{attribute 'qualified_only'}
VAR_GLOBAL CONSTANT
(* Super Mario Brothers Overworld *)
	NOTES_MAX : UINT := 3324;
	notes : ARRAY[0..NOTES_MAX] OF REAL := [146, 20, 0, 369, 20, 0, 659, 20, 47, 146, 20, 0, 369, 20, 0, 659, 20, 189, 146, 20, 0, 369, 20, 0, 659, 20, 190, 146, 20, 0, 369, 20, 0, 523, 20, 47, 146, 20, 0, 369, 20, 0, 659, 20, 190, 391, 20, 0, 493, 20, 0, 783, 20, 475, 195, 20, 0, 391, 20, 0, 195, 20, 0, 391, 20, 473, 195, 20, 0, 329, 20, 0, 523, 20, 332, 164, 20, 0, 261, 20, 0, 391, 20, 332, 130, 20, 0, 195, 20, 0, 329, 20, 332, 174, 20, 0, 261, 20, 0, 440, 20, 189, 195, 20, 0, 293, 20, 0, 493, 20, 189, 184, 20, 0, 277, 20, 0, 466, 20, 47, 174, 20, 0, 261, 20, 0, 440, 20, 190, 164, 20, 0, 261, 20, 0, 391, 20, 95, 261, 20, 0, 391, 20, 0, 659, 20, 95, 329, 20, 0, 493, 20, 0, 783, 20, 95, 349, 20, 0, 523, 20, 0, 880, 20, 190, 293, 20, 0, 440, 20, 0, 698, 20, 47, 329, 20, 0, 493, 20, 0, 783, 20, 189, 261, 20, 0, 440, 20, 0, 659, 20, 189, 220, 20, 0, 329, 20, 0, 523, 20, 47, 246, 20, 0, 349, 20, 0, 587, 20, 47, 195, 20, 0, 293, 20, 0, 493, 20, 332, 195, 20, 0, 329, 20, 0, 523, 20, 332, 164, 20, 0, 261, 20, 0, 391, 20, 332, 130, 20, 0, 195, 20, 0, 329, 20, 332, 174, 20, 0, 261, 20, 0, 440, 20, 189, 195, 20, 0, 293, 20, 0, 493, 20, 189, 184, 20, 0, 277, 20, 0, 466, 20, 47, 174, 20, 0, 261, 20, 0, 440, 20, 190, 164, 20, 0, 261, 20, 0, 391, 20, 95, 261, 20, 0, 391, 20, 0, 659, 20, 95, 329, 20, 0, 493, 20, 0, 783, 20, 95, 349, 20, 0, 523, 20, 0, 880, 20, 190, 293, 20, 0, 440, 20, 0, 698, 20, 47, 329, 20, 0, 493, 20, 0, 783, 20, 189, 261, 20, 0, 440, 20, 0, 659, 20, 189, 220, 20, 0, 329, 20, 0, 523, 20, 47, 246, 20, 0, 349, 20, 0, 587, 20, 47, 195, 20, 0, 293, 20, 0, 493, 20, 332, 130, 95, 190, 659, 20, 0, 783, 20, 0, 659, 20, 0, 783, 20, 47, 195, 20, 0, 622, 20, 0, 739, 20, 47, 587, 20, 0, 698, 20, 0, 587, 20, 0, 698, 20, 47, 493, 20, 0, 622, 20, 0, 493, 20, 0, 622, 20, 47, 261, 95, 47, 523, 20, 0, 659, 20, 0, 523, 20, 0, 659, 20, 47, 174, 95, 47, 329, 20, 0, 415, 20, 0, 329, 20, 0, 415, 20, 47, 349, 20, 0, 440, 20, 0, 349, 20, 0, 440, 20, 47, 261, 20, 0, 391, 20, 0, 523, 20, 47, 261, 95, 47, 261, 20, 0, 440, 20, 0, 261, 20, 0, 440, 20, 47, 174, 20, 0, 329, 20, 0, 523, 20, 47, 349, 20, 0, 587, 20, 0, 349, 20, 0, 587, 20, 47, 130, 95, 190, 659, 20, 0, 783, 20, 0, 659, 20, 0, 783, 20, 47, 164, 20, 0, 622, 20, 0, 739, 20, 47, 587, 20, 0, 698, 20, 0, 587, 20, 0, 698, 20, 47, 493, 20, 0, 622, 20, 0, 493, 20, 0, 622, 20, 47, 195, 95, 47, 261, 20, 0, 523, 20, 0, 659, 20, 189, 698, 20, 0, 783, 20, 0, 1046, 20, 189, 698, 20, 0, 783, 20, 0, 1046, 20, 47, 698, 20, 0, 783, 20, 0, 1046, 20, 190, 195, 95, 190, 130, 95, 190, 659, 20, 0, 783, 20, 0, 659, 20, 0, 783, 20, 47, 195, 20, 0, 622, 20, 0, 739, 20, 47, 587, 20, 0, 698, 20, 0, 587, 20, 0, 698, 20, 47, 493, 20, 0, 622, 20, 0, 493, 20, 0, 622, 20, 47, 261, 95, 47, 523, 20, 0, 659, 20, 0, 523, 20, 0, 659, 20, 47, 174, 95, 47, 329, 20, 0, 415, 20, 0, 329, 20, 0, 415, 20, 47, 349, 20, 0, 440, 20, 0, 349, 20, 0, 440, 20, 47, 261, 20, 0, 391, 20, 0, 523, 20, 47, 261, 95, 47, 261, 20, 0, 440, 20, 0, 261, 20, 0, 440, 20, 47, 174, 20, 0, 329, 20, 0, 523, 20, 47, 349, 20, 0, 587, 20, 0, 349, 20, 0, 587, 20, 47, 130, 95, 190, 207, 20, 0, 415, 20, 0, 622, 20, 332, 233, 20, 0, 349, 20, 0, 587, 20, 332, 261, 20, 0, 329, 20, 0, 523, 20, 332, 195, 94, 47, 195, 95, 190, 130, 95, 190, 130, 95, 190, 659, 20, 0, 783, 20, 0, 659, 20, 0, 783, 20, 47, 195, 20, 0, 622, 20, 0, 739, 20, 47, 587, 20, 0, 698, 20, 0, 587, 20, 0, 698, 20, 47, 493, 20, 0, 622, 20, 0, 493, 20, 0, 622, 20, 47, 261, 95, 47, 523, 20, 0, 659, 20, 0, 523, 20, 0, 659, 20, 47, 174, 95, 47, 329, 20, 0, 415, 20, 0, 329, 20, 0, 415, 20, 47, 349, 20, 0, 440, 20, 0, 349, 20, 0, 440, 20, 47, 261, 20, 0, 391, 20, 0, 523, 20, 47, 261, 95, 47, 261, 20, 0, 440, 20, 0, 261, 20, 0, 440, 20, 47, 174, 20, 0, 329, 20, 0, 523, 20, 47, 349, 20, 0, 587, 20, 0, 349, 20, 0, 587, 20, 47, 130, 95, 190, 659, 20, 0, 783, 20, 0, 659, 20, 0, 783, 20, 47, 164, 20, 0, 622, 20, 0, 739, 20, 47, 587, 20, 0, 698, 20, 0, 587, 20, 0, 698, 20, 47, 493, 20, 0, 622, 20, 0, 493, 20, 0, 622, 20, 47, 195, 95, 47, 261, 20, 0, 523, 20, 0, 659, 20, 189, 698, 20, 0, 783, 20, 0, 1046, 20, 189, 698, 20, 0, 783, 20, 0, 1046, 20, 47, 698, 20, 0, 783, 20, 0, 1046, 20, 190, 195, 95, 190, 130, 95, 190, 659, 20, 0, 783, 20, 0, 659, 20, 0, 783, 20, 47, 195, 20, 0, 622, 20, 0, 739, 20, 47, 587, 20, 0, 698, 20, 0, 587, 20, 0, 698, 20, 47, 493, 20, 0, 622, 20, 0, 493, 20, 0, 622, 20, 47, 261, 95, 47, 523, 20, 0, 659, 20, 0, 523, 20, 0, 659, 20, 47, 174, 95, 47, 329, 20, 0, 415, 20, 0, 329, 20, 0, 415, 20, 47, 349, 20, 0, 440, 20, 0, 349, 20, 0, 440, 20, 47, 261, 20, 0, 391, 20, 0, 523, 20, 47, 261, 95, 47, 261, 20, 0, 440, 20, 0, 261, 20, 0, 440, 20, 47, 174, 20, 0, 329, 20, 0, 523, 20, 47, 349, 20, 0, 587, 20, 0, 349, 20, 0, 587, 20, 47, 130, 95, 190, 207, 20, 0, 415, 20, 0, 622, 20, 332, 233, 20, 0, 349, 20, 0, 587, 20, 332, 261, 20, 0, 329, 20, 0, 523, 20, 332, 195, 94, 47, 195, 95, 190, 130, 95, 190, 103, 20, 0, 415, 20, 0, 523, 20, 47, 415, 20, 0, 523, 20, 0, 415, 20, 0, 523, 20, 189, 155, 20, 0, 415, 20, 0, 523, 20, 190, 415, 20, 0, 523, 20, 0, 415, 20, 0, 523, 20, 47, 207, 20, 0, 466, 20, 0, 587, 20, 190, 195, 20, 0, 391, 20, 0, 659, 20, 47, 329, 20, 0, 523, 20, 0, 329, 20, 0, 523, 20, 190, 130, 20, 0, 329, 20, 0, 440, 20, 47, 261, 20, 0, 391, 20, 0, 261, 20, 0, 391, 20, 189, 97, 95, 189, 103, 20, 0, 415, 20, 0, 523, 20, 47, 415, 20, 0, 523, 20, 0, 415, 20, 0, 523, 20, 189, 155, 20, 0, 415, 20, 0, 523, 20, 190, 415, 20, 0, 523, 20, 0, 415, 20, 0, 523, 20, 47, 207, 20, 0, 466, 20, 0, 587, 20, 47, 391, 20, 0, 659, 20, 0, 391, 20, 0, 659, 20, 47, 195, 95, 333, 130, 95, 332, 97, 95, 189, 103, 20, 0, 415, 20, 0, 523, 20, 47, 415, 20, 0, 523, 20, 0, 415, 20, 0, 523, 20, 189, 155, 20, 0, 415, 20, 0, 523, 20, 190, 415, 20, 0, 523, 20, 0, 415, 20, 0, 523, 20, 47, 207, 20, 0, 466, 20, 0, 587, 20, 190, 195, 20, 0, 391, 20, 0, 659, 20, 47, 329, 20, 0, 523, 20, 0, 329, 20, 0, 523, 20, 190, 130, 20, 0, 329, 20, 0, 440, 20, 47, 261, 20, 0, 391, 20, 0, 261, 20, 0, 391, 20, 189, 97, 95, 189, 146, 20, 0, 369, 20, 0, 659, 20, 47, 146, 20, 0, 369, 20, 0, 659, 20, 189, 146, 20, 0, 369, 20, 0, 659, 20, 190, 146, 20, 0, 369, 20, 0, 523, 20, 47, 146, 20, 0, 369, 20, 0, 659, 20, 190, 391, 20, 0, 493, 20, 0, 783, 20, 475, 195, 20, 0, 391, 20, 0, 195, 20, 0, 391, 20, 473, 195, 20, 0, 329, 20, 0, 523, 20, 332, 164, 20, 0, 261, 20, 0, 391, 20, 332, 130, 20, 0, 195, 20, 0, 329, 20, 332, 174, 20, 0, 261, 20, 0, 440, 20, 189, 195, 20, 0, 293, 20, 0, 493, 20, 189, 184, 20, 0, 277, 20, 0, 466, 20, 47, 174, 20, 0, 261, 20, 0, 440, 20, 190, 164, 20, 0, 261, 20, 0, 391, 20, 95, 261, 20, 0, 391, 20, 0, 659, 20, 95, 329, 20, 0, 493, 20, 0, 783, 20, 95, 349, 20, 0, 523, 20, 0, 880, 20, 190, 293, 20, 0, 440, 20, 0, 698, 20, 47, 329, 20, 0, 493, 20, 0, 783, 20, 189, 261, 20, 0, 440, 20, 0, 659, 20, 189, 220, 20, 0, 329, 20, 0, 523, 20, 47, 246, 20, 0, 349, 20, 0, 587, 20, 47, 195, 20, 0, 293, 20, 0, 493, 20, 332, 195, 20, 0, 329, 20, 0, 523, 20, 332, 164, 20, 0, 261, 20, 0, 391, 20, 332, 130, 20, 0, 195, 20, 0, 329, 20, 332, 174, 20, 0, 261, 20, 0, 440, 20, 189, 195, 20, 0, 293, 20, 0, 493, 20, 189, 184, 20, 0, 277, 20, 0, 466, 20, 47, 174, 20, 0, 261, 20, 0, 440, 20, 190, 164, 20, 0, 261, 20, 0, 391, 20, 95, 261, 20, 0, 391, 20, 0, 659, 20, 95, 329, 20, 0, 493, 20, 0, 783, 20, 95, 349, 20, 0, 523, 20, 0, 880, 20, 190, 293, 20, 0, 440, 20, 0, 698, 20, 47, 329, 20, 0, 493, 20, 0, 783, 20, 189, 261, 20, 0, 440, 20, 0, 659, 20, 189, 220, 20, 0, 329, 20, 0, 523, 20, 47, 246, 20, 0, 349, 20, 0, 587, 20, 47, 195, 20, 0, 293, 20, 0, 493, 20, 332, 130, 20, 0, 523, 20, 0, 659, 20, 47, 440, 20, 0, 523, 20, 0, 440, 20, 0, 523, 20, 190, 184, 20, 0, 329, 20, 0, 391, 20, 47, 195, 95, 190, 261, 20, 0, 329, 20, 0, 415, 20, 190, 174, 20, 0, 349, 20, 0, 440, 20, 47, 523, 20, 0, 698, 20, 0, 523, 20, 0, 698, 20, 47, 174, 95, 47, 523, 20, 0, 698, 20, 0, 523, 20, 0, 698, 20, 47, 261, 20, 0, 349, 20, 0, 440, 20, 47, 261, 94, 47, 174, 95, 190, 146, 20, 0, 391, 20, 0, 493, 20, 95, 698, 20, 0, 880, 20, 0, 698, 20, 0, 880, 20, 95, 698, 20, 0, 880, 20, 0, 174, 15, 0, 698, 15, 0, 880, 15, 0, 174, 47, 47, 195, 20, 0, 698, 20, 0, 880, 20, 95, 659, 20, 0, 783, 20, 0, 659, 20, 0, 783, 20, 0, 246, 95, 0, 587, 20, 0, 698, 20, 0, 587, 20, 0, 698, 20, 95, 195, 20, 0, 523, 20, 0, 659, 20, 47, 440, 20, 0, 523, 20, 0, 440, 20, 0, 523, 20, 47, 195, 95, 47, 349, 20, 0, 440, 20, 0, 349, 20, 0, 440, 20, 47, 261, 20, 0, 329, 20, 0, 391, 20, 47, 261, 94, 47, 195, 95, 190, 130, 20, 0, 523, 20, 0, 659, 20, 47, 440, 20, 0, 523, 20, 0, 440, 20, 0, 523, 20, 190, 184, 20, 0, 329, 20, 0, 391, 20, 47, 195, 95, 190, 261, 20, 0, 329, 20, 0, 415, 20, 190, 174, 20, 0, 349, 20, 0, 440, 20, 47, 523, 20, 0, 698, 20, 0, 523, 20, 0, 698, 20, 47, 174, 95, 47, 523, 20, 0, 698, 20, 0, 523, 20, 0, 698, 20, 47, 261, 20, 0, 349, 20, 0, 440, 20, 47, 261, 94, 47, 174, 95, 190, 195, 20, 0, 391, 20, 0, 493, 20, 47, 195, 20, 0, 587, 20, 0, 698, 20, 190, 195, 20, 0, 587, 20, 0, 698, 20, 47, 195, 20, 0, 587, 20, 0, 698, 20, 95, 220, 20, 0, 523, 20, 0, 659, 20, 95, 246, 20, 0, 493, 20, 0, 587, 20, 95, 261, 20, 0, 391, 20, 0, 523, 20, 47, 329, 95, 47, 195, 95, 47, 329, 95, 47, 130, 20, 0, 261, 20, 0, 130, 20, 0, 261, 20, 475, 130, 20, 0, 523, 20, 0, 659, 20, 47, 440, 20, 0, 523, 20, 0, 440, 20, 0, 523, 20, 190, 184, 20, 0, 329, 20, 0, 391, 20, 47, 195, 95, 190, 261, 20, 0, 329, 20, 0, 415, 20, 190, 174, 20, 0, 349, 20, 0, 440, 20, 47, 523, 20, 0, 698, 20, 0, 523, 20, 0, 698, 20, 47, 174, 95, 47, 523, 20, 0, 698, 20, 0, 523, 20, 0, 698, 20, 47, 261, 20, 0, 349, 20, 0, 440, 20, 47, 261, 94, 47, 174, 95, 190, 146, 20, 0, 391, 20, 0, 493, 20, 95, 698, 20, 0, 880, 20, 0, 698, 20, 0, 880, 20, 95, 698, 20, 0, 880, 20, 0, 174, 15, 0, 698, 15, 0, 880, 15, 0, 174, 47, 47, 195, 20, 0, 698, 20, 0, 880, 20, 95, 659, 20, 0, 783, 20, 0, 659, 20, 0, 783, 20, 0, 246, 95, 0, 587, 20, 0, 698, 20, 0, 587, 20, 0, 698, 20, 95, 195, 20, 0, 523, 20, 0, 659, 20, 47, 440, 20, 0, 523, 20, 0, 440, 20, 0, 523, 20, 47, 195, 95, 47, 349, 20, 0, 440, 20, 0, 349, 20, 0, 440, 20, 47, 261, 20, 0, 329, 20, 0, 391, 20, 47, 261, 94, 47, 195, 95, 190, 130, 20, 0, 523, 20, 0, 659, 20, 47, 440, 20, 0, 523, 20, 0, 440, 20, 0, 523, 20, 190, 184, 20, 0, 329, 20, 0, 391, 20, 47, 195, 95, 190, 261, 20, 0, 329, 20, 0, 415, 20, 190, 174, 20, 0, 349, 20, 0, 440, 20, 47, 523, 20, 0, 698, 20, 0, 523, 20, 0, 698, 20, 47, 174, 95, 47, 523, 20, 0, 698, 20, 0, 523, 20, 0, 698, 20, 47, 261, 20, 0, 349, 20, 0, 440, 20, 47, 261, 94, 47, 174, 95, 190, 195, 20, 0, 391, 20, 0, 493, 20, 47, 195, 20, 0, 587, 20, 0, 698, 20, 190, 195, 20, 0, 587, 20, 0, 698, 20, 47, 195, 20, 0, 587, 20, 0, 698, 20, 95, 220, 20, 0, 523, 20, 0, 659, 20, 95, 246, 20, 0, 493, 20, 0, 587, 20, 95, 261, 20, 0, 391, 20, 0, 523, 20, 47, 329, 95, 47, 195, 95, 47, 329, 95, 47, 130, 20, 0, 261, 20, 0, 130, 20, 0, 261, 20, 475, 103, 20, 0, 415, 20, 0, 523, 20, 47, 415, 20, 0, 523, 20, 0, 415, 20, 0, 523, 20, 189, 155, 20, 0, 415, 20, 0, 523, 20, 190, 415, 20, 0, 523, 20, 0, 415, 20, 0, 523, 20, 47, 207, 20, 0, 466, 20, 0, 587, 20, 190, 195, 20, 0, 391, 20, 0, 659, 20, 47, 329, 20, 0, 523, 20, 0, 329, 20, 0, 523, 20, 190, 130, 20, 0, 329, 20, 0, 440, 20, 47, 261, 20, 0, 391, 20, 0, 261, 20, 0, 391, 20, 189, 97, 95, 189, 103, 20, 0, 415, 20, 0, 523, 20, 47, 415, 20, 0, 523, 20, 0, 415, 20, 0, 523, 20, 189, 155, 20, 0, 415, 20, 0, 523, 20, 190, 415, 20, 0, 523, 20, 0, 415, 20, 0, 523, 20, 47, 207, 20, 0, 466, 20, 0, 587, 20, 47, 391, 20, 0, 659, 20, 0, 391, 20, 0, 659, 20, 47, 195, 95, 333, 130, 95, 332, 97, 95, 189, 103, 20, 0, 415, 20, 0, 523, 20, 47, 415, 20, 0, 523, 20, 0, 415, 20, 0, 523, 20, 189, 155, 20, 0, 415, 20, 0, 523, 20, 190, 415, 20, 0, 523, 20, 0, 415, 20, 0, 523, 20, 47, 207, 20, 0, 466, 20, 0, 587, 20, 190, 195, 20, 0, 391, 20, 0, 659, 20, 47, 329, 20, 0, 523, 20, 0, 329, 20, 0, 523, 20, 190, 130, 20, 0, 329, 20, 0, 440, 20, 47, 261, 20, 0, 391, 20, 0, 261, 20, 0, 391, 20, 189, 97, 95, 189, 146, 20, 0, 369, 20, 0, 659, 20, 47, 146, 20, 0, 369, 20, 0, 659, 20, 189, 146, 20, 0, 369, 20, 0, 659, 20, 190, 146, 20, 0, 369, 20, 0, 523, 20, 47, 146, 20, 0, 369, 20, 0, 659, 20, 190, 391, 20, 0, 493, 20, 0, 783, 20, 475, 195, 20, 0, 391, 20, 0, 195, 20, 0, 391, 20, 473, 130, 20, 0, 523, 20, 0, 659, 20, 47, 440, 20, 0, 523, 20, 0, 440, 20, 0, 523, 20, 190, 184, 20, 0, 329, 20, 0, 391, 20, 47, 195, 95, 190, 261, 20, 0, 329, 20, 0, 415, 20, 190, 174, 20, 0, 349, 20, 0, 440, 20, 47, 523, 20, 0, 698, 20, 0, 523, 20, 0, 698, 20, 47, 174, 95, 47, 523, 20, 0, 698, 20, 0, 523, 20, 0, 698, 20, 47, 261, 20, 0, 349, 20, 0, 440, 20, 47, 261, 94, 47, 174, 95, 190, 146, 20, 0, 391, 20, 0, 493, 20, 95, 698, 20, 0, 880, 20, 0, 698, 20, 0, 880, 20, 95, 698, 20, 0, 880, 20, 0, 174, 15, 0, 698, 15, 0, 880, 15, 0, 174, 47, 47, 195, 20, 0, 698, 20, 0, 880, 20, 95, 659, 20, 0, 783, 20, 0, 659, 20, 0, 783, 20, 0, 246, 95, 0, 587, 20, 0, 698, 20, 0, 587, 20, 0, 698, 20, 95, 195, 20, 0, 523, 20, 0, 659, 20, 47, 440, 20, 0, 523, 20, 0, 523, 20, 47, 195, 95, 47, 349, 20, 0, 440, 20, 0, 349, 20, 0, 440, 20, 47, 261, 20, 0, 329, 20, 0, 391, 20, 47, 261, 94, 47, 195, 95, 190, 130, 20, 0, 523, 20, 0, 659, 20, 47, 440, 20, 0, 523, 20, 0, 440, 20, 0, 523, 20, 190, 184, 20, 0, 329, 20, 0, 391, 20, 47, 195, 95, 190, 261, 20, 0, 329, 20, 0, 415, 20, 190, 174, 20, 0, 349, 20, 0, 440, 20, 47, 523, 20, 0, 698, 20, 0, 523, 20, 0, 698, 20, 47, 174, 95, 47, 523, 20, 0, 698, 20, 0, 523, 20, 0, 698, 20, 47, 261, 20, 0, 349, 20, 0, 440, 20, 47, 261, 94, 47, 174, 95, 190, 195, 20, 0, 391, 20, 0, 493, 20, 47, 195, 20, 0, 587, 20, 0, 698, 20, 190, 195, 20, 0, 587, 20, 0, 698, 20, 47, 195, 20, 0, 587, 20, 0, 698, 20, 95, 220, 20, 0, 523, 20, 0, 659, 20, 95, 246, 20, 0, 493, 20, 0, 587, 20, 95, 261, 20, 0, 391, 20, 0, 523, 20, 47, 329, 95, 47, 195, 95, 47, 329, 95, 47, 130, 20, 0, 261, 20, 0, 130, 20, 0, 261, 20, 0];
END_VAR

(* stored: Version 1.1.0.1, ProductVersion 3.1.4019.2
   GVL Mario: Id {d0910fa3-35c8-4f55-aabd-d14f02a63426} *)
